FUNCTION StartAction : bool
VAR_INPUT
	nom : STRING;
END_VAR
VAR
END_VAR

IF G_Match.Tableau[G_Match.iLigne].TypeAction = nom AND G_Match.iAsyncAction = '' 
OR G_Match.iAsyncAction = nom THEN
	G_Match.iAsyncAction := nom;
	StartAction := TRUE;
ELSE
	StartAction := FALSE;	
END_IF

END_FUNCTION

(* stored: Version 1.1.0.1, ProductVersion 3.1.4024.11
   POU StartAction: Id {78392568-e04f-442b-bc8a-ab460bb36abf}, SpecialFunc None *)
